// TwinCAT 3 PLC project PlcIotMqttv5ResSample
// ProgramVersion: 3.1.4020.4
// libraries:
//   Tc2_Standard, * (Beckhoff Automation GmbH)
//   Tc2_System, * (Beckhoff Automation GmbH)
//   Tc2_Utilities, * (Beckhoff Automation GmbH)
//   Tc3_IotBase, * (Beckhoff Automation GmbH)
//   Tc3_Module, * (Beckhoff Automation GmbH)
// project tree:
//   / PlcTask.TcTTO
//   POUs/ MAIN.TcPOU, PrgMqttCom.TcPOU
// (motion and I/O tree: see PLC project plciotmqttv5reqsample)
// real-time tasks:
//   TASK PlcTask: cycle T#10ms, priority 20, ADS port 350

CONFIGURATION PlcIotMqttv5ResSample
    RESOURCE PLC ON TwinCAT3
        TASK PlcTask(INTERVAL := T#10ms, PRIORITY := 20);
        PROGRAM MAIN WITH PlcTask : MAIN;
    END_RESOURCE
END_CONFIGURATION

// ---- POUs/MAIN.TcPOU
PROGRAM MAIN
VAR
END_VAR

PrgMqttCom();

END_PROGRAM

// ---- POUs/PrgMqttCom.TcPOU
(* This sample demonstrates the Request/Response mechanism of MQTTv5 as well as how to use UserProperties.
This PLC application will receive a request message from the broker and will send a response to the specified 
response topic. Please make sure that your message broker supports MQTTv5. *)
PROGRAM PrgMqttCom
VAR
	hrErrorOccurred	: HRESULT; // contains the latest occurred error
	hrPropRcv		: HRESULT;
	hrPropSet		: HRESULT;
	
	(* variable declarations for connection handling and set-up *)
	fbMqttClient	: FB_IotMqtt5Client;
	bSetParameter	: BOOL := TRUE; // if set to TRUE: sets connection parameters before connection establishment
	bConnect		: BOOL := TRUE; // if set to TRUE: starts connection establishment to message broker
	sReasonString	: STRING(255); // MQTTv5 Reason String property
	
	(* variable declarations for message handling, the message queue can be referenced directly from fbMqttClient output *)
	fbMessage		: FB_IotMqtt5Message;

	(* variable declarations for publish properties *)
	fbPubProps		: FB_IotMqtt5PublishProperties;
	sContentType	: STRING := 'my specific content';
	sName_User1		: STRING := 'Fritz';
	sValue_User1	: STRING := '68 kg';
	sName_User2		: STRING := 'Uwe';
	sValue_User2	: STRING := '76 kg';
	
	(* variable declarations for subscribe properties *)
	fbSubProps		: FB_IotMqtt5SubscribeProperties;

	(* variable declarations for ConnAck properties *)
	bRetainSupported : BOOL;

	(* request/response handling *)
	bSubscribedReq		: BOOL;			// if subscribed to the request
	nCorrDataRcvReq		: UDINT;
	sPayloadReq			: STRING(255) := 'HelloWorld';
	sPayloadRcv			: STRING(255);
	sPayloadRes			: STRING(255);
	sTopicReq			: STRING(255) := 'MyRequest';
	{attribute 'TcEncoding':='UTF-8'}
	sTopicRcv			: STRING(255);
	{attribute 'TcEncoding':='UTF-8'}
	sResponseTopicRcv	: STRING(255);
	{attribute 'TcEncoding':='UTF-8'}
	sContentTypeRcv		: STRING;
	aSubIdsRcv			: ARRAY[1..100] OF UDINT;
	i : UINT;
	aUserName_Rcv		: ARRAY[1..cMaxUserPropsToReceive] OF STRING;
	aUserValue_Rcv		: ARRAY[1..cMaxUserPropsToReceive] OF STRING;
	sValueByName		: STRING;
END_VAR
VAR CONSTANT
	cMaxUserPropsToReceive	: UINT := 20; // attend also Tc3_IotBase.ParameterList.cMaxMqtt5UserProps
END_VAR

// setting connection parameters once (broker address, port, TLS settings, ...)
IF bSetParameter THEN
	bSetParameter := FALSE;
	fbMqttClient.sHostName := 'localhost';
	fbMqttClient.nHostPort := 1883;
	
	// the following code snippet can be used if the message broker supports TLS
	(*
	fbMqttClient.nHostPort := 8883;
	fbMqttClient.stTLS.sCA := 'C:\TwinCAT\3.1\Target\Certificates\rootCA.pem';
	fbMqttClient.stTLS.sCert := 'C:\TwinCAT\3.1\Target\Certificates\myClientCert.pem';
	fbMqttClient.stTLS.sKeyFile := 'C:\TwinCAT\3.1\Target\Certificates\myClientPrivateKey.key';
	*) 
END_IF

// required: cyclic call of Execute method
fbMqttClient.Execute(bConnect);

// error handling
IF fbMqttClient.bError THEN
	// add your own error handling here
	hrErrorOccurred := fbMqttClient.hrErrorCode;
END_IF

// demonstrate usage of MQTTv5 ReasonString
IF NOT fbMqttClient.bConnected AND fbMqttClient.fbDisconnectProps.bPropertiesAvailable THEN
	sReasonString := fbMqttClient.fbDisconnectProps.sReasonString;
END_IF

// demonstrates how to access MQTTv5 ConnAckProperties
IF fbMqttClient.bConnected AND fbMqttClient.fbConnAckProps.bPropertiesAvailable THEN
	IF fbMqttClient.fbConnAckProps.bRetainAvailable THEN
		// Message Broker supports retain messages ...
		bRetainSupported := TRUE;
	END_IF
END_IF

// check if any messages have arrived
IF fbMqttClient.fbMessageQueue.nQueuedMessages > 0 THEN
	// a message has arrived -> retrieve the message from the queue and work with it
	IF fbMqttClient.fbMessageQueue.Dequeue(fbMessage:=fbMessage) THEN
		// get the topic on which the message has arrived
		fbMessage.GetTopic(pTopic:=ADR(sTopicRcv), nTopicSize:=SIZEOF(sTopicRcv) );	
		// if a message has been received on the response topic, then store the response in a variable (example)
		IF sTopicRcv = sTopicReq THEN
			// get payload from received message
			fbMessage.GetPayload(pPayload:=ADR(sPayloadRcv), nPayloadSize:=SIZEOF(sPayloadRcv), bSetNullTermination:=FALSE);
			// get requested response topic from received message
			hrPropRcv := fbMessage.GetResponseTopic(pResponseTopic:=ADR(sResponseTopicRcv), nResponseTopicSize:=SIZEOF(sResponseTopicRcv));
			// get correlation data from message and use it for the response so that sender can correlate the data
			IF SUCCEEDED(hrPropRcv) THEN		 
				hrPropRcv := fbMessage.GetCorrelationData(ADR(nCorrDataRcvReq), SIZEOF(nCorrDataRcvReq));
				IF SUCCEEDED(hrPropRcv) THEN
					// take payload that has been received in the request and re-use it in the response (just as an example) 
					sPayloadRes := CONCAT(sPayloadReq, TO_STRING(nCorrDataRcvReq));
					// response is sent on the response topic that has been specified as part of the request
				END_IF
			END_IF

			// get received publish properties
			sContentTypeRcv := fbMessage.sContentType;
			IF SUCCEEDED(hrPropRcv) AND fbMessage.nSubIdCnt > 0 THEN
				hrPropRcv := fbMessage.GetSubIds(aSubIds:=aSubIdsRcv);
			END_IF

			// get all UserProperties from message
			IF fbMessage.nUserPropertyCnt > 0 THEN
				FOR i := 1 TO MIN(fbMessage.nUserPropertyCnt, cMaxUserPropsToReceive) DO
					IF SUCCEEDED(hrPropRcv) THEN
						hrPropRcv := fbMessage.GetUserPropertyByIdx(nIdx:=i-1, pName:=ADR(aUserName_Rcv[i]), nNameSize:=SIZEOF(aUserName_Rcv[i]), pValue:=ADR(aUserValue_Rcv[i]), nValueSize:=SIZEOF(aUserValue_Rcv[i]) );
					END_IF
				END_FOR
			END_IF

			// get a specific UserProperty from message
			IF SUCCEEDED(hrPropRcv) THEN
				hrPropRcv := fbMessage.GetUserPropertyValueByName(sName := 'Uwe', pValue:=ADR(sValueByName), nValueSize:=SIZEOF(sValueByName) );
			END_IF

			// set PublishProperties for response
			fbPubProps.sContentType := sContentType;
			fbPubProps.nMsgExpiryInterval := 7;
			fbPubProps.bTopicAlias := TRUE;
			fbPubProps.bPayloadUtf8 := TRUE;
			fbPubProps.ClearUserProperties();
			
			// add UserProperties to PublishProperties
			hrPropSet := fbPubProps.AddUserProperty(sName_User1, sValue_User1);
			hrPropSet := fbPubProps.AddUserProperty(sName_User2, sValue_User2);
			
			// send response using the requested response topic and the prepared response message
			fbMqttClient.Response(	sResponseTopic:= sResponseTopicRcv, 
									pPayload:= ADR(sPayloadRes), nPayloadSize:= LEN2(ADR(sPayloadRes))+1, 
									eQoS:= TcIotMqttQos.AtMostOnceDelivery, bRetain:= FALSE, bQueue:= FALSE, 
									pProps:=fbPubProps.pPublishProperties, pCorrelationData:=ADR(nCorrDataRcvReq), nCorrelationDataSize:=SIZEOF(nCorrDataRcvReq) );
															
			// error handling
			IF fbMqttClient.bError THEN
				// add your own error handling here
				hrErrorOccurred := fbMqttClient.hrErrorCode;
			END_IF
		END_IF
	END_IF
END_IF

// execute the following code only when connected to the message broker
IF fbMqttClient.bConnected THEN
	// check if a subscription has been created to the request topic. If not, create it.
	IF NOT bSubscribedReq THEN
		// set a SubID
		fbSubProps.nSubId := 17;
		// subscribe to request topic
		bSubscribedReq := fbMqttClient.Subscribe(sTopic:=sTopicReq, eQoS:=TcIotMqttQos.AtMostOnceDelivery, pProps:=fbSubProps.pSubscribeProperties);
		// error handling
		IF fbMqttClient.bError THEN
			// add your own error handling here
			hrErrorOccurred := fbMqttClient.hrErrorCode;
		END_IF
	END_IF
END_IF

END_PROGRAM
